// TIA Portal V19 export
DATA_BLOCK "DB_Variantenbefehl"   // DB43
{ S7_Optimized_Access := 'FALSE' }
// stored: AutoNumber false
   VAR RETAIN
      Anzahl_Varianten : Int := 1;   // vorläufige Platzhaltervariable
      Offset : Int := 10;   // Beginn der Daten
      max_Var : Int := 6;   // maximale Anzahl von Varianten (ENTSPRICHT DER FELDLÄNGE)
      resW : Int := 0;
      resW1 : Int := 0;
      Variante : Array[0..1] of Struct
         Pos : Array[1..6] of Byte;
      END_STRUCT;
   END_VAR
BEGIN
   Variante[0].Pos[1] := 16#16;
   Variante[0].Pos[2] := 16#13;
   Variante[0].Pos[3] := 16#11;
   Variante[0].Pos[4] := 16#0E;
   Variante[0].Pos[5] := 16#0D;
   Variante[0].Pos[6] := 16#0A;
   Variante[1].Pos[1..6] := 16#00;
END_DATA_BLOCK
